PROGRAM Stn055_PrgCalls
VAR
END_VAR

//Turn on the default programs
IF gFirstScan THEN
	gDebug_ComponentCalls.CallStn055_21_StorageBreakStopsRed := TRUE;
	gDebug_ComponentCalls.CallStn055_40_StorageBypassDivertRed := TRUE;
	gDebug_ComponentCalls.CallStn055_41_StorageBypassMainMergePrestopRed := TRUE;
	gDebug_ComponentCalls.CallStn055_42_StorageBypassSpurMergePrestopRed := TRUE;
	gDebug_ComponentCalls.CallStn055_43_StorageBypassMergeRed := TRUE;
	gDebug_ComponentCalls.CallStn055_45_Stn511Divert := TRUE;
	gDebug_ComponentCalls.CallStn055_46_Stn511MainMergePrestop := TRUE;
	gDebug_ComponentCalls.CallStn055_47_Stn511Merge := TRUE;
	gDebug_ComponentCalls.CallStn055_50_Stn512Divert := TRUE;
	gDebug_ComponentCalls.CallStn055_51_Stn512MainMergePrestop := TRUE;
	gDebug_ComponentCalls.CallStn055_52_Stn512Merge := TRUE;
	
	gDebug_ComponentCalls.CallStn055_20_StorageBreakStopsGrn := TRUE;
	gDebug_ComponentCalls.CallStn055_25_StorageBypassDivertGrn := TRUE;
	gDebug_ComponentCalls.CallStn055_26_StorageBypassMainMergePrestopGrn  := TRUE;
	gDebug_ComponentCalls.CallStn055_27_StorageBypassSpurMergePrestopGrn := TRUE;
	gDebug_ComponentCalls.CallStn055_28_StorageBypassMergeGrn := TRUE;
	gDebug_ComponentCalls.CallStn055_30_Stn411Divert := TRUE;
	gDebug_ComponentCalls.CallStn055_31_Stn411MainMergePrestop := TRUE;
	gDebug_ComponentCalls.CallStn055_32_Stn411Merge := TRUE;
	
END_IF

// Call Components
IF gDebug_ComponentCalls.CallStn055_20_StorageBreakStopsGrn OR
		gFirstScan THEN
	Stn055_20_StorageBreakStopsGrn();
END_IF
IF gDebug_ComponentCalls.CallStn055_21_StorageBreakStopsRed OR
		gFirstScan THEN
	Stn055_21_StorageBreakStopsRed();
END_IF
IF gDebug_ComponentCalls.CallStn055_25_StorageBypassDivertGrn OR
		gFirstScan THEN
	Stn055_25_StorageBypassDivertGrn();
END_IF
IF gDebug_ComponentCalls.CallStn055_26_StorageBypassMainMergePrestopGrn OR
		gFirstScan THEN
	Stn055_26_StorageBypassMainMergePrestopGrn();
END_IF
IF gDebug_ComponentCalls.CallStn055_27_StorageBypassSpurMergePrestopGrn OR
		gFirstScan THEN
	Stn055_27_StorageBypassSpurMergePrestopGrn();
END_IF
IF gDebug_ComponentCalls.CallStn055_28_StorageBypassMergeGrn OR
		gFirstScan THEN
	Stn055_28_StorageBypassMergeGrn();
END_IF
IF gDebug_ComponentCalls.CallStn055_30_Stn411Divert OR
		gFirstScan THEN
	Stn055_30_Stn411Divert();
END_IF
IF gDebug_ComponentCalls.CallStn055_31_Stn411MainMergePrestop OR
		gFirstScan THEN
	Stn055_31_Stn411MainMergePrestop();
END_IF
IF gDebug_ComponentCalls.CallStn055_32_Stn411Merge OR
		gFirstScan THEN
	Stn055_32_Stn411Merge();
END_IF
IF gDebug_ComponentCalls.CallStn055_40_StorageBypassDivertRed OR
		gFirstScan THEN
	Stn055_40_StorageBypassDivertRed();
END_IF
IF gDebug_ComponentCalls.CallStn055_41_StorageBypassMainMergePrestopRed OR
		gFirstScan THEN
	Stn055_41_StorageBypassMainMergePrestopRed();
END_IF
IF gDebug_ComponentCalls.CallStn055_42_StorageBypassSpurMergePrestopRed OR
		gFirstScan THEN
	Stn055_42_StorageBypassSpurMergePrestopRed();
END_IF
IF gDebug_ComponentCalls.CallStn055_43_StorageBypassMergeRed OR
		gFirstScan THEN
	Stn055_43_StorageBypassMergeRed();
END_IF
IF gDebug_ComponentCalls.CallStn055_45_Stn511Divert OR
		gFirstScan THEN
	Stn055_45_Stn511Divert();
END_IF
IF gDebug_ComponentCalls.CallStn055_46_Stn511MainMergePrestop OR
		gFirstScan THEN
	Stn055_46_Stn511MainMergePrestop();
END_IF
IF gDebug_ComponentCalls.CallStn055_47_Stn511Merge OR
		gFirstScan THEN
	Stn055_47_Stn511Merge();
END_IF
IF gDebug_ComponentCalls.CallStn055_50_Stn512Divert OR
		gFirstScan THEN
	Stn055_50_Stn512Divert();
END_IF
IF gDebug_ComponentCalls.CallStn055_51_Stn512MainMergePrestop OR
		gFirstScan THEN
	Stn055_51_Stn512MainMergePrestop();
END_IF
IF gDebug_ComponentCalls.CallStn055_52_Stn512Merge OR
		gFirstScan THEN
	Stn055_52_Stn512Merge();
END_IF

END_PROGRAM

(* stored: Version 1.1.0.1, ProductVersion 3.1.4024.6
   POU Stn055_PrgCalls: Id {c24ade0f-2287-4d00-b38b-3cd15669f233}, SpecialFunc None *)
